FUNCTION_BLOCK FB_ThirdObject
VAR_INPUT
END_VAR
VAR_OUTPUT
END_VAR
VAR
	_parentObject : ITF_Object;
END_VAR

METHOD FB_init : BOOL
VAR_INPUT
	bInitRetains : BOOL; // if TRUE, the retain variables are initialized (warm start / cold start)
	bInCopyCode : BOOL;  // if TRUE, the instance afterwards gets moved into the copy code (online change)
	ParentObject : ITF_Object;
END_VAR
_parentObject := ParentObject;
END_METHOD

END_FUNCTION_BLOCK

(* stored: Version 1.1.0.1, ProductVersion 3.1.4024.11
   POU FB_ThirdObject: Id {cf740e6b-86ed-48db-b106-663968cd5241}, SpecialFunc None
   Method FB_init: Id {f32fca7e-b31d-43a0-ad58-d0162a78c803} *)
